FUNCTION_BLOCK Test IMPLEMENTS I_TestOperation
VAR
	_TestId		: T_MaxString;
	_State		: E_TestStatus;
	TestMessage : FB_TcMessage;
    Source      : FB_TcSourceInfo;
END_VAR

METHOD AssertEqual
VAR_INPUT
	Expected : ANY;
	Actual	 : ANY;
	Epsilon	 : LREAL := 0.000001;
END_VAR

VAR
	nCount		   : DINT;
	StringExpected : T_MaxString;
	StringActual   : T_MaxString;
	LrealExpected  : LREAL;
	LrealActual	   : LREAL;
	RealExpected   : REAL;
	RealActual	   : REAL;
END_VAR
IF Expected.typeclass <> Actual.typeclass THEN
	State := E_TestStatus.DoneFailed;
	ReportAssert('Type missmatch!');
	RETURN;
END_IF

IF Expected.diSize <> Actual.diSize THEN
	State := E_TestStatus.DoneFailed;
	ReportAssert('Type size missmatch!');
	RETURN;
END_IF

// String
IF Expected.TypeClass = __SYSTEM.TYPE_CLASS.TYPE_ANYSTRING OR Expected.TypeClass = __SYSTEM.TYPE_CLASS.TYPE_STRING OR Expected.TypeClass = __SYSTEM.TYPE_CLASS.TYPE_WSTRING OR Expected.TypeClass = __SYSTEM.TYPE_CLASS.TYPE_XSTRING THEN
	MEMCPY(destAddr := ADR(StringExpected), srcAddr := Expected.pValue, n := DINT_TO_UDINT(Expected.diSize));
	MEMCPY(destAddr := ADR(StringActual), srcAddr := Actual.pValue, n := DINT_TO_UDINT(Actual.diSize));
	IF StringExpected <> StringActual THEN
		State := E_TestStatus.DoneFailed;
		ReportAssert(CONCAT(CONCAT('Expected: ', GetValueString(Expected)), CONCAT(' , Actual: ', GetValueString(Actual))));
		RETURN;
	END_IF
ELSIF Expected.TypeClass = __SYSTEM.TYPE_CLASS.TYPE_LREAL THEN
	MEMCPY(destAddr := ADR(LrealExpected), srcAddr := Expected.pValue, n := DINT_TO_UDINT(Expected.diSize));
	MEMCPY(destAddr := ADR(LrealActual), srcAddr := Actual.pValue, n := DINT_TO_UDINT(Actual.diSize));
	IF ((LrealExpected - Epsilon) > LrealActual) OR ((LrealExpected + Epsilon) < LrealActual) THEN
		State := E_TestStatus.DoneFailed;
		ReportAssert(CONCAT(CONCAT('Expected: ', GetValueString(Expected)), CONCAT(' , Actual: ', GetValueString(Actual))));
		RETURN;
	END_IF
ELSIF Expected.TypeClass = __SYSTEM.TYPE_CLASS.TYPE_ANYREAL OR Expected.TypeClass = __SYSTEM.TYPE_CLASS.TYPE_REAL THEN
	MEMCPY(destAddr := ADR(RealExpected), srcAddr := Expected.pValue, n := DINT_TO_UDINT(Expected.diSize));
	MEMCPY(destAddr := ADR(RealActual), srcAddr := Actual.pValue, n := DINT_TO_UDINT(Actual.diSize));
	IF ((RealExpected - Epsilon) > RealActual) OR ((RealExpected + Epsilon) < RealActual) THEN
		State := E_TestStatus.DoneFailed;
		ReportAssert(CONCAT(CONCAT('Expected: ', GetValueString(Expected)), CONCAT(' , Actual: ', GetValueString(Actual))));
		RETURN;
	END_IF
ELSE
	// Byte comparison
	FOR nCount := 0 TO Actual.diSize - 1 DO
		IF Expected.pvalue[nCount] <> Actual.pvalue[nCount] THEN
			State := E_TestStatus.DoneFailed;
			ReportAssert(CONCAT(CONCAT('Expected: ', GetValueString(Expected)), CONCAT(' , Actual: ', GetValueString(Actual))));
			RETURN;
		END_IF
	END_FOR
END_IF

State := E_TestStatus.DoneOk;
END_METHOD

METHOD ExecuteTest : BOOL
VAR_INPUT
END_VAR
IF State = E_TestStatus.Init THEN
	State := E_TestStatus.Running;
END_IF

ExecuteTest := State = E_TestStatus.Running;
END_METHOD

METHOD PRIVATE ReportAssert
VAR_INPUT
	Reason : STRING := '';
END_VAR

VAR
	ResultString : T_MaxString;
END_VAR
Source.sName := 'Test Suite';
TestMessage.Create(eventClass	:= TC_EVENT_CLASSES.TestEvents,
				   nEventId		:= 1,
				   eSeverity	:= TcEventSeverity.Error,
				   ipSourceInfo := 0);

ResultString := CONCAT('Test failed - ', TestId);
ResultString := CONCAT(ResultString, '! ');
ResultString := CONCAT(ResultString, Reason);
TestMessage.ipArguments.AddString(ResultString);
TestMessage.Send(0);
Source.Clear();
END_METHOD

PROPERTY State :  E_TestStatus
GET
State := _State;
END_GET
SET
_State := State;
END_SET
END_PROPERTY

PROPERTY TestId : T_MaxString
GET
TestId := _TestId;
END_GET
SET
_TestId := TestId;
END_SET
END_PROPERTY

END_FUNCTION_BLOCK

(* stored: Version 1.1.0.1
   POU Test: Id {9e8aece1-ee26-4cf6-b4f4-25a27cfed9dc}, SpecialFunc None
   Method AssertEqual: Id {848da2d4-fc83-435a-a497-3700fbb8f173}
   Method ExecuteTest: Id {d3490801-b397-4b9a-8a9d-6332802fd972}
   Method ReportAssert: Id {70613942-8c38-478a-ad8e-0d3b3e114371}
   Property State: Id {107dda4b-11bf-4131-8c5f-64011be55284}
   Get Get: Id {262d28c9-71be-4402-bd2c-a86901ea6f86}
   Set Set: Id {71ba93ec-d3d4-4f07-892c-f28b00d83612}
   Property TestId: Id {0723af9d-7a0b-479f-bfbc-daf60795c791}
   Get Get: Id {b9dea5fd-624e-4410-bf21-8a9d9c1236f8}
   Set Set: Id {b3f6ef0d-a7cd-4254-a831-4165b3f53021} *)
